(* PLC project OpenPLC, Unknown OpenPLC 1 *)
(* stored: creationDateTime 2026-02-21T00:00:00, modificationDateTime 2026-02-21T00:00:00 *)

TYPE STATION_T : STRUCT
  number : INT;
  x_mm : REAL;
  station_type : INT;
  device_delay_s : REAL;
  dropping_time_s : REAL;
END_STRUCT;
END_TYPE

TYPE PHYSICS_2D_T : STRUCT
  x_accel_s : REAL;
  x_decel_s : REAL;
  x_max_mm_s : REAL;
  z_total_mm : REAL;
  z_slow_dry_mm : REAL;
  z_slow_wet_mm : REAL;
  z_slow_end_mm : REAL;
  z_slow_mm_s : REAL;
  z_fast_mm_s : REAL;
  drip_delay_s : REAL;
  avoid_mm : REAL;
END_STRUCT;
END_TYPE

TYPE TRANSPORTER_CFG_T : STRUCT
  id : INT;
  start_station : INT;
  x_min_limit : REAL;
  x_max_limit : REAL;
  phys2d : PHYSICS_2D_T;
END_STRUCT;
END_TYPE

TYPE TRANSPORTER_STATE_T : STRUCT
  active : BOOL;
  phase : INT;
  z_stage : INT;
  x_mm : REAL;
  z_mm : REAL;
  vel_x : REAL;
  vel_z : REAL;
  current_station : INT;
  lift_station_target : INT;
  sink_station_target : INT;
  target_x : REAL;
  x_min_limit : REAL;
  x_max_limit : REAL;
  z_timer_s : REAL;
END_STRUCT;
END_TYPE

FUNCTION IsWetStationType : BOOL
  VAR_INPUT
    station_type : INT;
  END_VAR

            IsWetStationType := (station_type = 1) OR (station_type = 11);
          
END_FUNCTION

FUNCTION FindStationIndexByNumber : INT
  VAR_INPUT
    station_number : INT;
  END_VAR
  VAR
    i : INT;
    tmp_st : STATION_T;
  END_VAR

            FindStationIndexByNumber := 0;
FOR i := 1 TO g_station_count DO
  tmp_st := g_stations[i];
  IF tmp_st.number = station_number THEN
    FindStationIndexByNumber := i;
    RETURN;
  END_IF;
END_FOR;
          
END_FUNCTION

FUNCTION GetStationX : REAL
  VAR_INPUT
    station_number : INT;
  END_VAR
  VAR
    idx : INT;
    tmp_st : STATION_T;
  END_VAR

            idx := FindStationIndexByNumber(station_number);
IF idx > 0 THEN
  tmp_st := g_stations[idx];
  GetStationX := tmp_st.x_mm;
ELSE
  GetStationX := 0.0;
END_IF;
          
END_FUNCTION

FUNCTION GetStationType : INT
  VAR_INPUT
    station_number : INT;
  END_VAR
  VAR
    idx : INT;
    tmp_st : STATION_T;
  END_VAR

            idx := FindStationIndexByNumber(station_number);
IF idx > 0 THEN
  tmp_st := g_stations[idx];
  GetStationType := tmp_st.station_type;
ELSE
  GetStationType := 0;
END_IF;
          
END_FUNCTION

FUNCTION GetStationDeviceDelay : REAL
  VAR_INPUT
    station_number : INT;
  END_VAR
  VAR
    idx : INT;
    tmp_st : STATION_T;
  END_VAR

            idx := FindStationIndexByNumber(station_number);
IF idx > 0 THEN
  tmp_st := g_stations[idx];
  GetStationDeviceDelay := tmp_st.device_delay_s;
ELSE
  GetStationDeviceDelay := 0.0;
END_IF;
          
END_FUNCTION

FUNCTION GetStationDroppingTime : REAL
  VAR_INPUT
    station_number : INT;
  END_VAR
  VAR
    idx : INT;
    tmp_st : STATION_T;
  END_VAR

            idx := FindStationIndexByNumber(station_number);
IF idx > 0 THEN
  tmp_st := g_stations[idx];
  GetStationDroppingTime := tmp_st.dropping_time_s;
ELSE
  GetStationDroppingTime := 0.0;
END_IF;
          
END_FUNCTION

FUNCTION_BLOCK FB_XMotion
  VAR_INPUT
    delta_t : REAL;
    x_target : REAL;
    x_min : REAL;
    x_max : REAL;
    v_max : REAL;
    t_acc : REAL;
    t_dec : REAL;
  END_VAR
  VAR_IN_OUT
    x_pos : REAL;
    v_x : REAL;
  END_VAR
  VAR_OUTPUT
    arrived : BOOL;
  END_VAR
  VAR
    drive_target : REAL;
    distance : REAL;
    dir : REAL;
    a_acc : REAL;
    a_dec : REAL;
    brake_dist : REAL;
    new_vel : REAL;
    travel : REAL;
  END_VAR

            IF (x_max > x_min) THEN
  IF x_pos < x_min THEN
    drive_target := x_min;
  ELSIF x_pos > x_max THEN
    drive_target := x_max;
  ELSE
    IF x_target < x_min THEN
      drive_target := x_min;
    ELSIF x_target > x_max THEN
      drive_target := x_max;
    ELSE
      drive_target := x_target;
    END_IF;
  END_IF;
ELSE
  drive_target := x_target;
END_IF;

arrived := ABS(x_pos - drive_target) <= 3.0;
IF arrived THEN
  x_pos := drive_target;
  v_x := 0.0;
  RETURN;
END_IF;

IF t_acc <= 0.0 THEN t_acc := 0.001; END_IF;
IF t_dec <= 0.0 THEN t_dec := 0.001; END_IF;
IF v_max < 0.0 THEN v_max := 0.0; END_IF;

a_acc := v_max / t_acc;
a_dec := v_max / t_dec;

dir := 1.0;
IF drive_target < x_pos THEN
  dir := -1.0;
END_IF;

distance := ABS(drive_target - x_pos);

IF a_dec > 0.0 THEN
  brake_dist := (v_x * v_x) / (2.0 * a_dec);
ELSE
  brake_dist := 0.0;
END_IF;

IF brake_dist >= distance THEN
  new_vel := v_x - a_dec * delta_t;
  IF new_vel < 0.0 THEN new_vel := 0.0; END_IF;
ELSE
  new_vel := v_x + a_acc * delta_t;
  IF new_vel > v_max THEN new_vel := v_max; END_IF;
END_IF;

travel := new_vel * delta_t;
  IF travel >= distance THEN
    x_pos := drive_target;
    v_x := 0.0;
    arrived := TRUE;
  ELSE
    x_pos := x_pos + dir * travel;
    v_x := new_vel;
    arrived := FALSE;
  END_IF;
          
END_FUNCTION_BLOCK

PROGRAM PLC_PRG
  VAR
    init_done : BOOL := FALSE;
    i : INT;
    idx : INT;
    station_type : INT;
    device_delay : REAL;
    drop_time : REAL;
    slow_start : REAL;
    arrived_x : BOOL;
    nearest_num : INT;
    min_dist : REAL;
    dx : REAL;
    fb_x : ARRAY[1..10] OF FB_XMotion;
  END_VAR

            IF NOT init_done THEN
  g_station_count := 21;

  g_stations[1] := (number := 101, x_mm := 100.0, station_type := 22, device_delay_s := 0.0, dropping_time_s := 0.0);
  g_stations[2] := (number := 102, x_mm := 1550.0, station_type := 30, device_delay_s := 0.0, dropping_time_s := 0.0);
  g_stations[3] := (number := 103, x_mm := 3000.0, station_type := 30, device_delay_s := 0.0, dropping_time_s := 0.0);
  g_stations[4] := (number := 104, x_mm := 4450.0, station_type := 0, device_delay_s := 3.0, dropping_time_s := 0.0);
  g_stations[5] := (number := 105, x_mm := 5900.0, station_type := 0, device_delay_s := 3.0, dropping_time_s := 0.0);
  g_stations[6] := (number := 106, x_mm := 7350.0, station_type := 0, device_delay_s := 3.0, dropping_time_s := 0.0);
  g_stations[7] := (number := 107, x_mm := 8800.0, station_type := 1, device_delay_s := 3.0, dropping_time_s := 10.0);
  g_stations[8] := (number := 108, x_mm := 10250.0, station_type := 1, device_delay_s := 0.0, dropping_time_s := 10.0);
  g_stations[9] := (number := 109, x_mm := 11700.0, station_type := 1, device_delay_s := 0.0, dropping_time_s := 10.0);
  g_stations[10] := (number := 110, x_mm := 13150.0, station_type := 1, device_delay_s := 0.0, dropping_time_s := 10.0);
  g_stations[11] := (number := 111, x_mm := 14600.0, station_type := 1, device_delay_s := 0.0, dropping_time_s := 10.0);
  g_stations[12] := (number := 112, x_mm := 16050.0, station_type := 1, device_delay_s := 3.0, dropping_time_s := 10.0);
  g_stations[13] := (number := 113, x_mm := 17500.0, station_type := 1, device_delay_s := 0.0, dropping_time_s := 10.0);
  g_stations[14] := (number := 114, x_mm := 18950.0, station_type := 32, device_delay_s := 0.0, dropping_time_s := 0.0);
  g_stations[15] := (number := 115, x_mm := 20400.0, station_type := 0, device_delay_s := 3.0, dropping_time_s := 10.0);
  g_stations[16] := (number := 116, x_mm := 21850.0, station_type := 1, device_delay_s := 3.0, dropping_time_s := 10.0);
  g_stations[17] := (number := 117, x_mm := 23300.0, station_type := 1, device_delay_s := 0.0, dropping_time_s := 10.0);
  g_stations[18] := (number := 118, x_mm := 24750.0, station_type := 1, device_delay_s := 0.0, dropping_time_s := 10.0);
  g_stations[19] := (number := 119, x_mm := 26200.0, station_type := 30, device_delay_s := 0.0, dropping_time_s := 0.0);
  g_stations[20] := (number := 120, x_mm := 27650.0, station_type := 30, device_delay_s := 0.0, dropping_time_s := 0.0);
  g_stations[21] := (number := 121, x_mm := 29100.0, station_type := 1, device_delay_s := 0.0, dropping_time_s := 10.0);

  g_cfg[1].id := 1;
  g_cfg[1].start_station := 101;
  g_cfg[1].x_min_limit := 100.0;
  g_cfg[1].x_max_limit := 20600.0;
  g_cfg[1].phys2d := (
    x_accel_s := 1.5,
    x_decel_s := 1.5,
    x_max_mm_s := 500.0,
    z_total_mm := 2500.0,
    z_slow_dry_mm := 300.0,
    z_slow_wet_mm := 1000.0,
    z_slow_end_mm := 50.0,
    z_slow_mm_s := 100.0,
    z_fast_mm_s := 200.0,
    drip_delay_s := 5.0,
    avoid_mm := 2000.0
  );

  g_cfg[2].id := 2;
  g_cfg[2].start_station := 118;
  g_cfg[2].x_min_limit := 14300.0;
  g_cfg[2].x_max_limit := 29100.0;
  g_cfg[2].phys2d := (
    x_accel_s := 1.5,
    x_decel_s := 1.5,
    x_max_mm_s := 500.0,
    z_total_mm := 2500.0,
    z_slow_dry_mm := 300.0,
    z_slow_wet_mm := 1000.0,
    z_slow_end_mm := 50.0,
    z_slow_mm_s := 100.0,
    z_fast_mm_s := 200.0,
    drip_delay_s := 5.0,
    avoid_mm := 2000.0
  );

  FOR i := 1 TO MAX_TRANSPORTERS DO
    g_state[i].active := (i <= 2);
    g_state[i].phase := PHASE_IDLE;
    g_state[i].z_stage := Z_IDLE;
    g_state[i].vel_x := 0.0;
    g_state[i].vel_z := 0.0;
    g_state[i].z_timer_s := 0.0;
    g_state[i].x_min_limit := g_cfg[i].x_min_limit;
    g_state[i].x_max_limit := g_cfg[i].x_max_limit;

    idx := FindStationIndexByNumber(g_cfg[i].start_station);
    IF idx > 0 THEN
      g_state[i].x_mm := g_stations[idx].x_mm;
      g_state[i].current_station := g_stations[idx].number;
    ELSE
      g_state[i].x_mm := 0.0;
      g_state[i].current_station := 0;
    END_IF;
    g_state[i].z_mm := 0.0;
  END_FOR;

  init_done := TRUE;
END_IF;

FOR i := 1 TO MAX_TRANSPORTERS DO
  IF NOT g_state[i].active THEN
    CONTINUE;
  END_IF;

  IF (g_state[i].phase = PHASE_IDLE) AND g_cmd_start[i] THEN
    g_state[i].lift_station_target := g_cmd_lift_station[i];
    g_state[i].sink_station_target := g_cmd_sink_station[i];
    g_state[i].target_x := GetStationX(g_state[i].lift_station_target);
    g_state[i].phase := PHASE_MOVE_TO_LIFT;
    g_state[i].z_stage := Z_IDLE;
    g_state[i].z_timer_s := 0.0;
  END_IF;

  IF g_state[i].phase = PHASE_MOVE_TO_LIFT THEN
    fb_x[i](
      delta_t := DT_S,
      x_target := g_state[i].target_x,
      x_min := g_state[i].x_min_limit,
      x_max := g_state[i].x_max_limit,
      v_max := g_cfg[i].phys2d.x_max_mm_s,
      t_acc := g_cfg[i].phys2d.x_accel_s,
      t_dec := g_cfg[i].phys2d.x_decel_s,
      x_pos := g_state[i].x_mm,
      v_x := g_state[i].vel_x
    );
    arrived_x := fb_x[i].arrived;
    IF arrived_x THEN
      g_state[i].current_station := g_state[i].lift_station_target;
      device_delay := GetStationDeviceDelay(g_state[i].lift_station_target);
      drop_time := GetStationDroppingTime(g_state[i].lift_station_target);
      g_state[i].z_timer_s := device_delay + drop_time;
      g_state[i].z_stage := Z_DELAY_UP;
      g_state[i].phase := PHASE_LIFTING;
    END_IF;
  END_IF;

  IF g_state[i].phase = PHASE_LIFTING THEN
    station_type := GetStationType(g_state[i].lift_station_target);
    IF IsWetStationType(station_type) THEN
      slow_start := g_cfg[i].phys2d.z_slow_wet_mm;
    ELSE
      slow_start := g_cfg[i].phys2d.z_slow_dry_mm;
    END_IF;

    CASE g_state[i].z_stage OF
      Z_DELAY_UP:
        g_state[i].z_timer_s := g_state[i].z_timer_s - DT_S;
        IF g_state[i].z_timer_s <= 0.0 THEN
          g_state[i].z_stage := Z_UP_SLOW;
          g_state[i].z_mm := g_cfg[i].phys2d.z_total_mm;
        END_IF;
      Z_UP_SLOW:
        g_state[i].z_mm := g_state[i].z_mm - g_cfg[i].phys2d.z_slow_mm_s * DT_S;
        IF g_state[i].z_mm <= (g_cfg[i].phys2d.z_total_mm - slow_start) THEN
          g_state[i].z_stage := Z_UP_FAST;
        END_IF;
      Z_UP_FAST:
        g_state[i].z_mm := g_state[i].z_mm - g_cfg[i].phys2d.z_fast_mm_s * DT_S;
        IF g_state[i].z_mm <= g_cfg[i].phys2d.z_slow_end_mm THEN
          g_state[i].z_stage := Z_UP_SLOW_END;
        END_IF;
      Z_UP_SLOW_END:
        g_state[i].z_mm := g_state[i].z_mm - g_cfg[i].phys2d.z_slow_mm_s * DT_S;
        IF g_state[i].z_mm <= 0.0 THEN
          g_state[i].z_mm := 0.0;
          g_state[i].z_timer_s := g_cfg[i].phys2d.drip_delay_s;
          g_state[i].z_stage := Z_DRIP_UP;
        END_IF;
      Z_DRIP_UP:
        g_state[i].z_timer_s := g_state[i].z_timer_s - DT_S;
        IF g_state[i].z_timer_s <= 0.0 THEN
          g_state[i].z_stage := Z_IDLE;
          g_state[i].target_x := GetStationX(g_state[i].sink_station_target);
          g_state[i].phase := PHASE_MOVE_TO_SINK;
        END_IF;
    ELSE
    END_CASE;
  END_IF;

  IF g_state[i].phase = PHASE_MOVE_TO_SINK THEN
    fb_x[i](
      delta_t := DT_S,
      x_target := g_state[i].target_x,
      x_min := g_state[i].x_min_limit,
      x_max := g_state[i].x_max_limit,
      v_max := g_cfg[i].phys2d.x_max_mm_s,
      t_acc := g_cfg[i].phys2d.x_accel_s,
      t_dec := g_cfg[i].phys2d.x_decel_s,
      x_pos := g_state[i].x_mm,
      v_x := g_state[i].vel_x
    );
    arrived_x := fb_x[i].arrived;
    IF arrived_x THEN
      g_state[i].current_station := g_state[i].sink_station_target;
      device_delay := GetStationDeviceDelay(g_state[i].sink_station_target);
      g_state[i].z_timer_s := device_delay + g_cfg[i].phys2d.drip_delay_s;
      g_state[i].z_stage := Z_DELAY_DOWN;
      g_state[i].phase := PHASE_SINKING;
    END_IF;
  END_IF;

  IF g_state[i].phase = PHASE_SINKING THEN
    station_type := GetStationType(g_state[i].sink_station_target);
    IF IsWetStationType(station_type) THEN
      slow_start := g_cfg[i].phys2d.z_slow_wet_mm;
    ELSE
      slow_start := g_cfg[i].phys2d.z_slow_dry_mm;
    END_IF;

    CASE g_state[i].z_stage OF
      Z_DELAY_DOWN:
        g_state[i].z_timer_s := g_state[i].z_timer_s - DT_S;
        IF g_state[i].z_timer_s <= 0.0 THEN
          g_state[i].z_stage := Z_DOWN_FAST;
        END_IF;
      Z_DOWN_FAST:
        g_state[i].z_mm := g_state[i].z_mm + g_cfg[i].phys2d.z_fast_mm_s * DT_S;
        IF g_state[i].z_mm >= (g_cfg[i].phys2d.z_total_mm - slow_start) THEN
          g_state[i].z_stage := Z_DOWN_SLOW;
        END_IF;
      Z_DOWN_SLOW:
        g_state[i].z_mm := g_state[i].z_mm + g_cfg[i].phys2d.z_slow_mm_s * DT_S;
        IF g_state[i].z_mm >= g_cfg[i].phys2d.z_total_mm THEN
          g_state[i].z_mm := g_cfg[i].phys2d.z_total_mm;
          g_state[i].z_stage := Z_IDLE;
          g_state[i].phase := PHASE_IDLE;
        END_IF;
    ELSE
    END_CASE;
  END_IF;

  min_dist := 1.0e9;
  nearest_num := g_state[i].current_station;
  FOR idx := 1 TO g_station_count DO
    dx := g_stations[idx].x_mm - g_state[i].x_mm;
    IF ABS(dx) < min_dist THEN
      min_dist := ABS(dx);
      nearest_num := g_stations[idx].number;
    END_IF;
  END_FOR;
  g_state[i].current_station := nearest_num;
END_FOR;
          
END_PROGRAM

CONFIGURATION Config0
  VAR_GLOBAL CONSTANT
    MAX_TRANSPORTERS : INT := 10;
    MAX_STATIONS : INT := 21;
    DT_S : REAL := 0.02;
    PHASE_IDLE : INT := 0;
    PHASE_MOVE_TO_LIFT : INT := 1;
    PHASE_LIFTING : INT := 2;
    PHASE_MOVE_TO_SINK : INT := 3;
    PHASE_SINKING : INT := 4;
    Z_IDLE : INT := 0;
    Z_DELAY_UP : INT := 1;
    Z_UP_SLOW : INT := 2;
    Z_UP_FAST : INT := 3;
    Z_UP_SLOW_END : INT := 4;
    Z_DRIP_UP : INT := 5;
    Z_DELAY_DOWN : INT := 6;
    Z_DOWN_FAST : INT := 7;
    Z_DOWN_SLOW : INT := 8;
  END_VAR
  VAR_GLOBAL
    g_station_count : INT := 0;
    g_stations : ARRAY[1..21] OF STATION_T;
    g_cfg : ARRAY[1..10] OF TRANSPORTER_CFG_T;
    g_state : ARRAY[1..10] OF TRANSPORTER_STATE_T;
    g_cmd_start : ARRAY[1..10] OF BOOL;
    g_cmd_lift_station : ARRAY[1..10] OF INT;
    g_cmd_sink_station : ARRAY[1..10] OF INT;
  END_VAR
  RESOURCE Res0 ON PLC
    TASK task0(INTERVAL := T#20ms, PRIORITY := 0);
    PROGRAM instance0 WITH task0 : PLC_PRG;
  END_RESOURCE
END_CONFIGURATION
